TYPE Vec5i : ARRAY[1..5] OF INT; END_TYPE

(* stored: Version 1.1.0.1, ProductVersion 3.1.4024.12
   DUT Vec5i: Id {cc5dc7b9-3e18-4d3f-9aa7-baf832eb7fb6} *)
